FUNCTION_BLOCK "Unit_FC_Sub"
{ S7_Optimized_Access := 'TRUE' }
VERSION : 0.1
   VAR
      a { ExternalAccessible := 'False'; ExternalVisible := 'False'; ExternalWritable := 'False'} : Bool;
   END_VAR

   VAR_TEMP
      _ret : Bool;
   END_VAR


BEGIN
	"BeforeEach"(iName:= GetBlockName(DINT#15));


	#_ret := "assertEqualsINT"(actual:= "FC_Sub"(i1:= int#5, i2:= int#10),expected:= int#-5);
	#_ret := "assertEqualsINT"(actual:= "FC_Sub"(i1:= int#10, i2:= int#10),expected:= int#0);


	"AfterEach"();


END_FUNCTION_BLOCK

